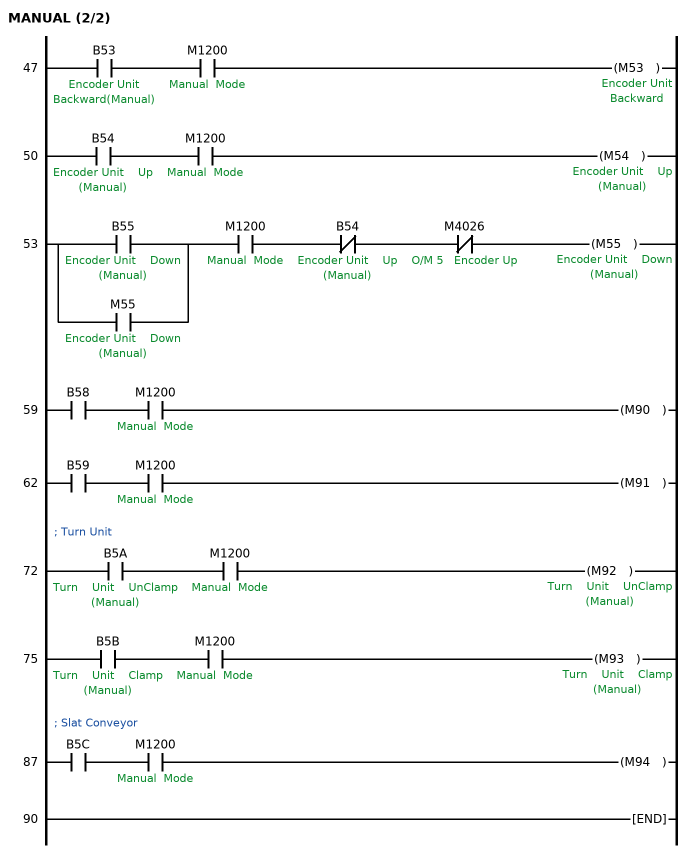
[picture p24: ladder of MANUAL, rungs at steps 47 to 90]
47    LD      B53  ; Encoder Unit    Backward(Manual)
      AND     M1200  ; Manual  Mode
      OUT     M53  ; Encoder Unit    Backward
50    LD      B54  ; Encoder Unit    Up      (Manual)
      AND     M1200  ; Manual  Mode
      OUT     M54  ; Encoder Unit    Up      (Manual)
53    LD      B55  ; Encoder Unit    Down    (Manual)
      OR      M55  ; Encoder Unit    Down    (Manual)
      AND     M1200  ; Manual  Mode
      ANI     B54  ; Encoder Unit    Up      (Manual)
      ANI     M4026  ; O/M 5   Encoder Up
      OUT     M55  ; Encoder Unit    Down    (Manual)
59    LD      B58
      AND     M1200  ; Manual  Mode
      OUT     M90
62    LD      B59
      AND     M1200  ; Manual  Mode
      OUT     M91
; Turn Unit
72    LD      B5A  ; Turn    Unit    UnClamp (Manual)
      AND     M1200  ; Manual  Mode
      OUT     M92  ; Turn    Unit    UnClamp (Manual)
75    LD      B5B  ; Turn    Unit    Clamp   (Manual)
      AND     M1200  ; Manual  Mode
      OUT     M93  ; Turn    Unit    Clamp   (Manual)
; Slat Conveyor
87    LD      B5C
      AND     M1200  ; Manual  Mode
      OUT     M94
90    END
END_PROGRAM

PROGRAM ORIGIN
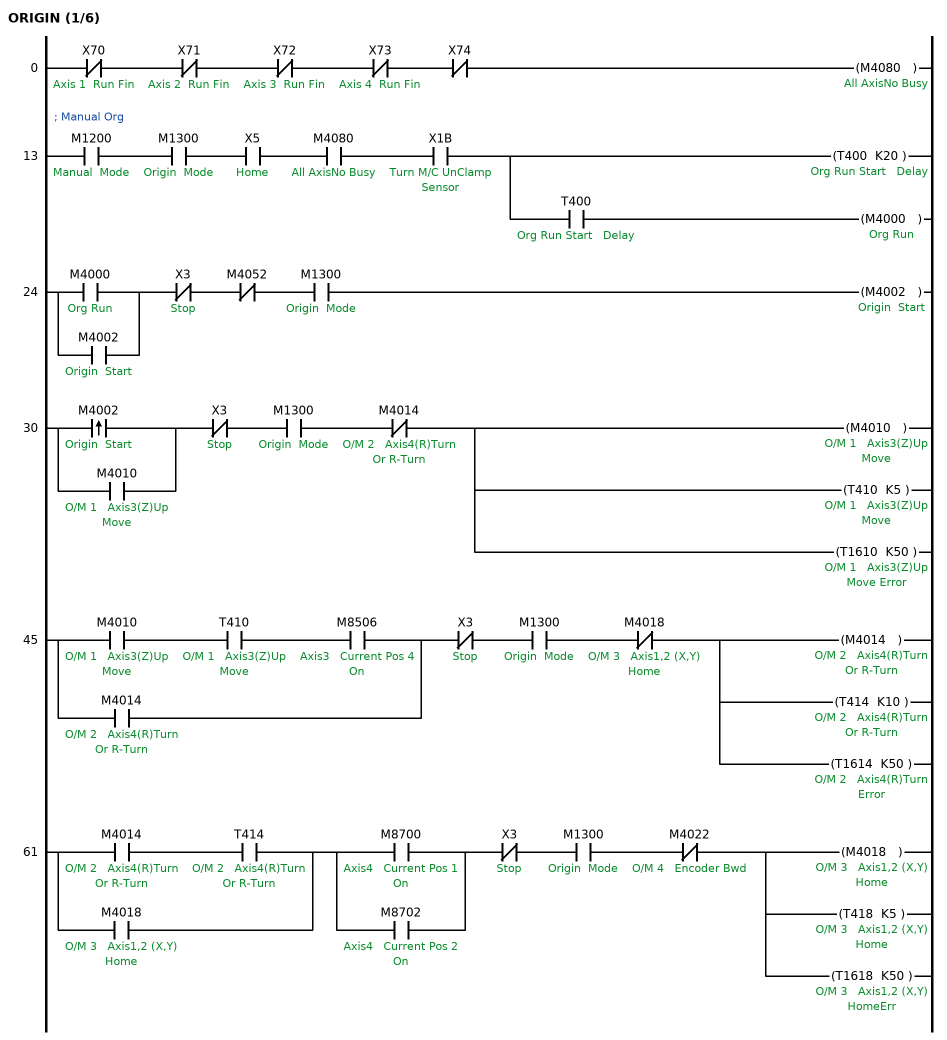
0     LDI     X70  ; Axis 1  Run Fin
      ANI     X71  ; Axis 2  Run Fin
      ANI     X72  ; Axis 3  Run Fin
      ANI     X73  ; Axis 4  Run Fin
      ANI     X74
      OUT     M4080  ; All AxisNo Busy
; Manual Org
13    LD      M1200  ; Manual  Mode
      AND     M1300  ; Origin  Mode
      AND     X5  ; Home
      AND     M4080  ; All AxisNo Busy
      AND     X1B  ; Turn M/C UnClamp Sensor
      OUT     T400 K20  ; Org Run Start   Delay
      AND     T400  ; Org Run Start   Delay
      OUT     M4000  ; Org Run
24    LD      M4000  ; Org Run
      OR      M4002  ; Origin  Start
      ANI     X3  ; Stop
      ANI     M4052
      AND     M1300  ; Origin  Mode
      OUT     M4002  ; Origin  Start
30    LDP     M4002  ; Origin  Start
      OR      M4010  ; O/M 1   Axis3(Z)Up Move
      ANI     X3  ; Stop
      AND     M1300  ; Origin  Mode
      ANI     M4014  ; O/M 2   Axis4(R)Turn Or R-Turn
      OUT     M4010  ; O/M 1   Axis3(Z)Up Move
      OUT     T410 K5  ; O/M 1   Axis3(Z)Up Move
      OUT     T1610 K50  ; O/M 1   Axis3(Z)Up Move Error
45    LD      M4010  ; O/M 1   Axis3(Z)Up Move
      AND     T410  ; O/M 1   Axis3(Z)Up Move
      AND     M8506  ; Axis3   Current Pos 4 On
      OR      M4014  ; O/M 2   Axis4(R)Turn Or R-Turn
      ANI     X3  ; Stop
      AND     M1300  ; Origin  Mode
      ANI     M4018  ; O/M 3   Axis1,2 (X,Y)   Home
      OUT     M4014  ; O/M 2   Axis4(R)Turn Or R-Turn
      OUT     T414 K10  ; O/M 2   Axis4(R)Turn Or R-Turn
      OUT     T1614 K50  ; O/M 2   Axis4(R)Turn    Error
61    LD      M4014  ; O/M 2   Axis4(R)Turn Or R-Turn
      AND     T414  ; O/M 2   Axis4(R)Turn Or R-Turn
      OR      M4018  ; O/M 3   Axis1,2 (X,Y)   Home
      LD      M8700  ; Axis4   Current Pos 1 On
      OR      M8702  ; Axis4   Current Pos 2 On
      ANB
      ANI     X3  ; Stop
      AND     M1300  ; Origin  Mode
      ANI     M4022  ; O/M 4   Encoder Bwd
      OUT     M4018  ; O/M 3   Axis1,2 (X,Y)   Home
      OUT     T418 K5  ; O/M 3   Axis1,2 (X,Y)   Home
      OUT     T1618 K50  ; O/M 3   Axis1,2 (X,Y)   HomeErr
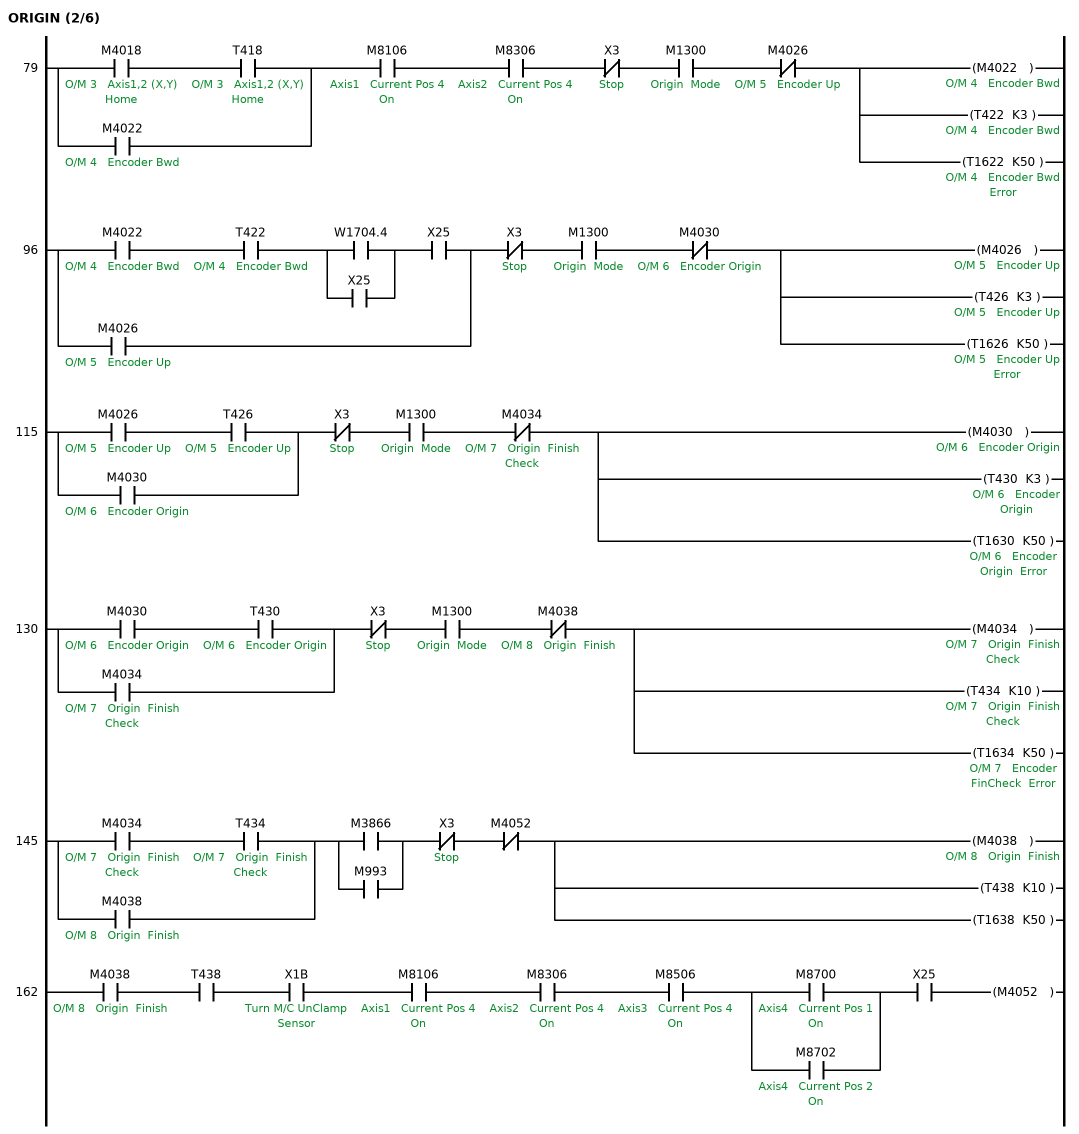
79    LD      M4018  ; O/M 3   Axis1,2 (X,Y)   Home
      AND     T418  ; O/M 3   Axis1,2 (X,Y)   Home
      OR      M4022  ; O/M 4   Encoder Bwd
      AND     M8106  ; Axis1   Current Pos 4 On
      AND     M8306  ; Axis2   Current Pos 4 On
      ANI     X3  ; Stop
      AND     M1300  ; Origin  Mode
      ANI     M4026  ; O/M 5   Encoder Up
      OUT     M4022  ; O/M 4   Encoder Bwd
      OUT     T422 K3  ; O/M 4   Encoder Bwd
      OUT     T1622 K50  ; O/M 4   Encoder Bwd     Error
96    LD      M4022  ; O/M 4   Encoder Bwd
      AND     T422  ; O/M 4   Encoder Bwd
      LD      W1704.4
      OR      X25
      ANB
      AND     X25
      OR      M4026  ; O/M 5   Encoder Up
      ANI     X3  ; Stop
      AND     M1300  ; Origin  Mode
      ANI     M4030  ; O/M 6   Encoder Origin
      OUT     M4026  ; O/M 5   Encoder Up
      OUT     T426 K3  ; O/M 5   Encoder Up
      OUT     T1626 K50  ; O/M 5   Encoder Up      Error
115   LD      M4026  ; O/M 5   Encoder Up
      AND     T426  ; O/M 5   Encoder Up
      OR      M4030  ; O/M 6   Encoder Origin
      ANI     X3  ; Stop
      AND     M1300  ; Origin  Mode
      ANI     M4034  ; O/M 7   Origin  Finish  Check
      OUT     M4030  ; O/M 6   Encoder Origin
      OUT     T430 K3  ; O/M 6   Encoder Origin
      OUT     T1630 K50  ; O/M 6   Encoder Origin  Error
130   LD      M4030  ; O/M 6   Encoder Origin
      AND     T430  ; O/M 6   Encoder Origin
      OR      M4034  ; O/M 7   Origin  Finish  Check
      ANI     X3  ; Stop
      AND     M1300  ; Origin  Mode
      ANI     M4038  ; O/M 8   Origin  Finish
      OUT     M4034  ; O/M 7   Origin  Finish  Check
      OUT     T434 K10  ; O/M 7   Origin  Finish  Check
      OUT     T1634 K50  ; O/M 7   Encoder FinCheck  Error
145   LD      M4034  ; O/M 7   Origin  Finish  Check
      AND     T434  ; O/M 7   Origin  Finish  Check
      OR      M4038  ; O/M 8   Origin  Finish
      LD      M3866
      OR      M993
      ANB
      ANI     X3  ; Stop
      ANI     M4052
      OUT     M4038  ; O/M 8   Origin  Finish
      OUT     T438 K10
      OUT     T1638 K50
162   LD      M4038  ; O/M 8   Origin  Finish
      AND     T438
      AND     X1B  ; Turn M/C UnClamp Sensor
      AND     M8106  ; Axis1   Current Pos 4 On
      AND     M8306  ; Axis2   Current Pos 4 On
      AND     M8506  ; Axis3   Current Pos 4 On
      LD      M8700  ; Axis4   Current Pos 1 On
      OR      M8702  ; Axis4   Current Pos 2 On
      ANB
      AND     X25
      OUT     M4052
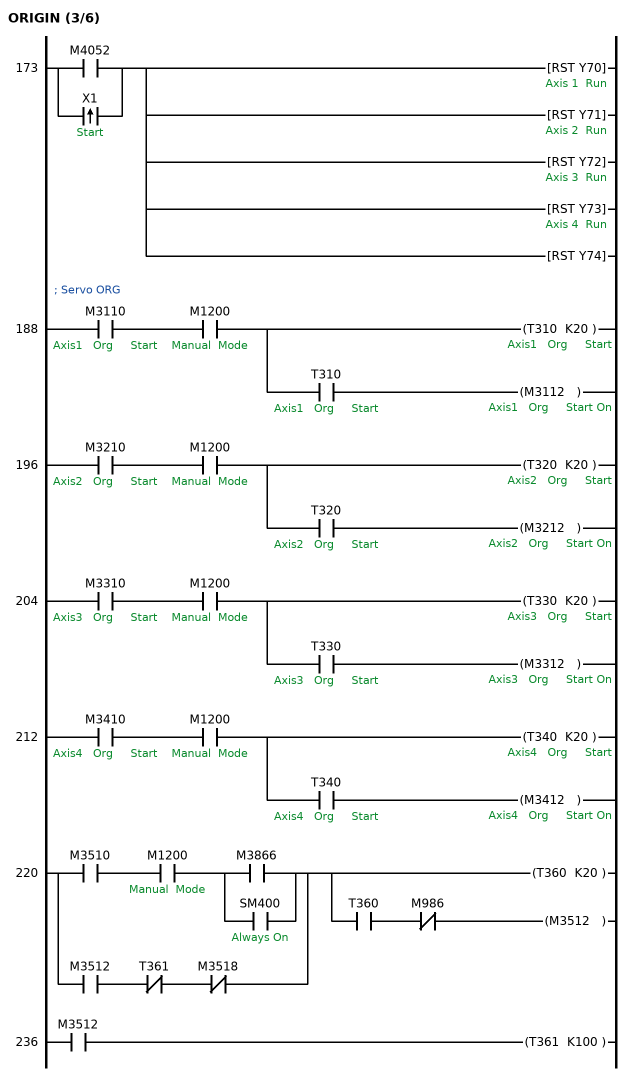
173   LD      M4052
      ORP     X1  ; Start
      RST     Y70  ; Axis 1  Run
      RST     Y71  ; Axis 2  Run
      RST     Y72  ; Axis 3  Run
      RST     Y73  ; Axis 4  Run
      RST     Y74
; Servo ORG
188   LD      M3110  ; Axis1   Org     Start
      AND     M1200  ; Manual  Mode
      OUT     T310 K20  ; Axis1   Org     Start
      AND     T310  ; Axis1   Org     Start
      OUT     M3112  ; Axis1   Org     Start On
196   LD      M3210  ; Axis2   Org     Start
      AND     M1200  ; Manual  Mode
      OUT     T320 K20  ; Axis2   Org     Start
      AND     T320  ; Axis2   Org     Start
      OUT     M3212  ; Axis2   Org     Start On
204   LD      M3310  ; Axis3   Org     Start
      AND     M1200  ; Manual  Mode
      OUT     T330 K20  ; Axis3   Org     Start
      AND     T330  ; Axis3   Org     Start
      OUT     M3312  ; Axis3   Org     Start On
212   LD      M3410  ; Axis4   Org     Start
      AND     M1200  ; Manual  Mode
      OUT     T340 K20  ; Axis4   Org     Start
      AND     T340  ; Axis4   Org     Start
      OUT     M3412  ; Axis4   Org     Start On
220   LD      M3510
      AND     M1200  ; Manual  Mode
      LD      M3866
      OR      SM400  ; Always On
      ANB
      LD      M3512
      ANI     T361
      ANI     M3518
      ORB
      OUT     T360 K20
      AND     T360
      ANI     M986
      OUT     M3512
236   LD      M3512
      OUT     T361 K100
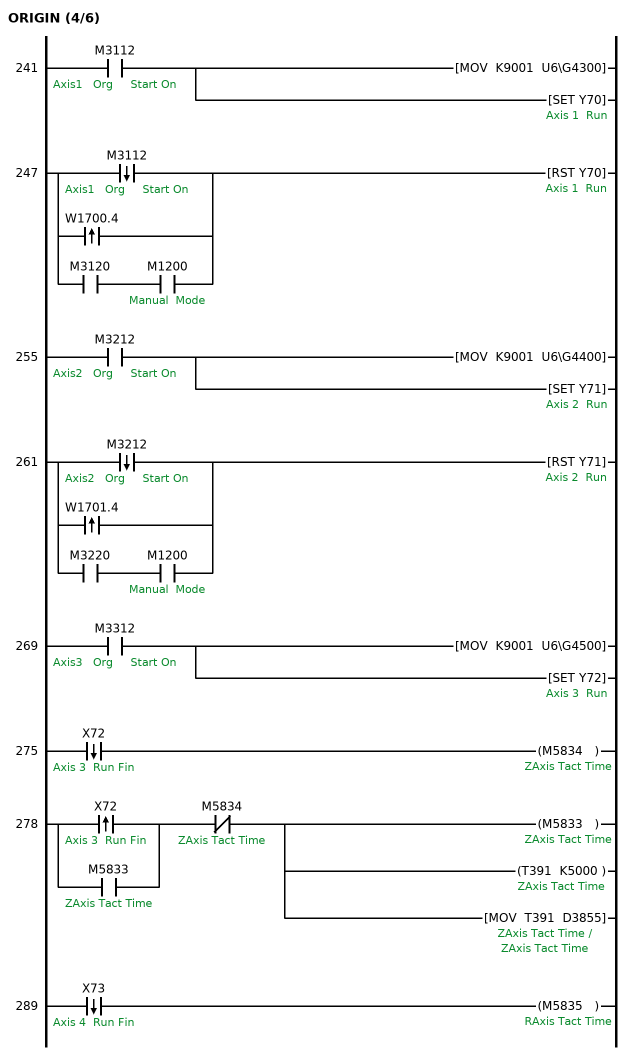
241   LD      M3112  ; Axis1   Org     Start On
      MOV     K9001 U6\G4300
      SET     Y70  ; Axis 1  Run
247   LDF     M3112  ; Axis1   Org     Start On
      ORP     W1700.4
      LD      M3120
      AND     M1200  ; Manual  Mode
      ORB
      RST     Y70  ; Axis 1  Run
255   LD      M3212  ; Axis2   Org     Start On
      MOV     K9001 U6\G4400
      SET     Y71  ; Axis 2  Run
261   LDF     M3212  ; Axis2   Org     Start On
      ORP     W1701.4
      LD      M3220
      AND     M1200  ; Manual  Mode
      ORB
      RST     Y71  ; Axis 2  Run
269   LD      M3312  ; Axis3   Org     Start On
      MOV     K9001 U6\G4500
      SET     Y72  ; Axis 3  Run
275   LDF     X72  ; Axis 3  Run Fin
      OUT     M5834  ; ZAxis Tact Time
278   LDP     X72  ; Axis 3  Run Fin
      OR      M5833  ; ZAxis Tact Time
      ANI     M5834  ; ZAxis Tact Time
      OUT     M5833  ; ZAxis Tact Time
      OUT     T391 K5000  ; ZAxis Tact Time
      MOV     T391 D3855  ; ZAxis Tact Time
289   LDF     X73  ; Axis 4  Run Fin
      OUT     M5835  ; RAxis Tact Time
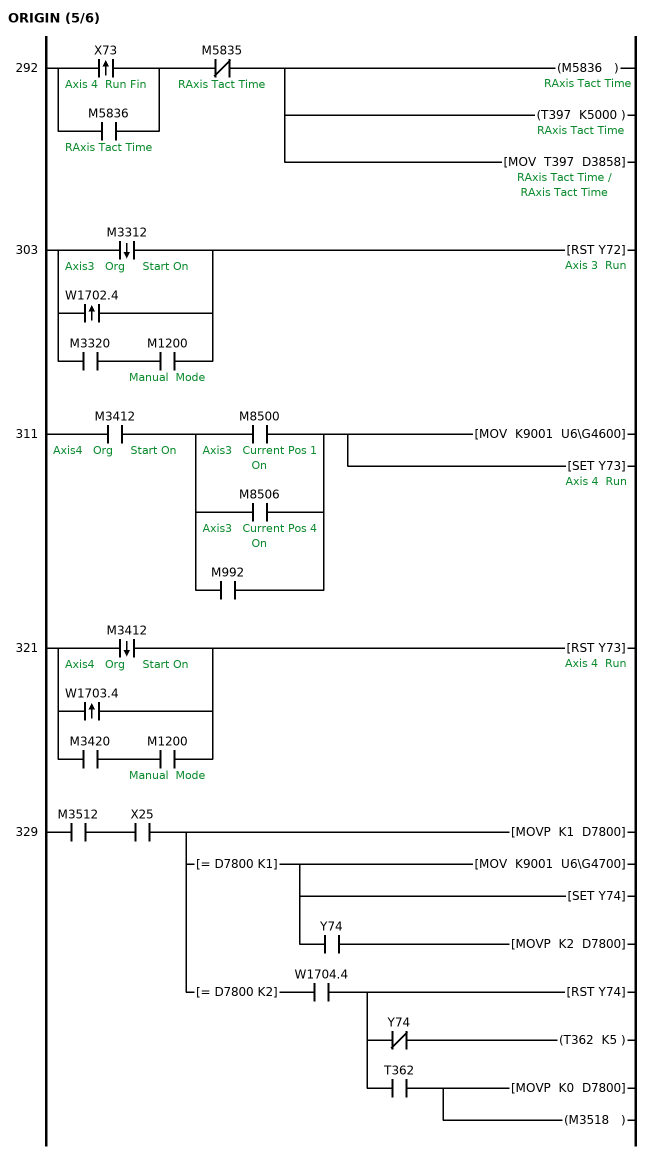
292   LDP     X73  ; Axis 4  Run Fin
      OR      M5836  ; RAxis Tact Time
      ANI     M5835  ; RAxis Tact Time
      OUT     M5836  ; RAxis Tact Time
      OUT     T397 K5000  ; RAxis Tact Time
      MOV     T397 D3858  ; RAxis Tact Time
303   LDF     M3312  ; Axis3   Org     Start On
      ORP     W1702.4
      LD      M3320
      AND     M1200  ; Manual  Mode
      ORB
      RST     Y72  ; Axis 3  Run
311   LD      M3412  ; Axis4   Org     Start On
      LD      M8500  ; Axis3   Current Pos 1 On
      OR      M8506  ; Axis3   Current Pos 4 On
      OR      M992
      ANB
      MOV     K9001 U6\G4600
      SET     Y73  ; Axis 4  Run
321   LDF     M3412  ; Axis4   Org     Start On
      ORP     W1703.4
      LD      M3420
      AND     M1200  ; Manual  Mode
      ORB
      RST     Y73  ; Axis 4  Run
329   LD      M3512
      AND     X25
      MOVP    K1 D7800
      MPS
      AND=    D7800 K1
      MOV     K9001 U6\G4700
      SET     Y74
      AND     Y74
      MOVP    K2 D7800
      MPP
      AND=    D7800 K2
      AND     W1704.4
      RST     Y74
      MPS
      ANI     Y74
      OUT     T362 K5
      MPP
      AND     T362
      MOVP    K0 D7800
      OUT     M3518
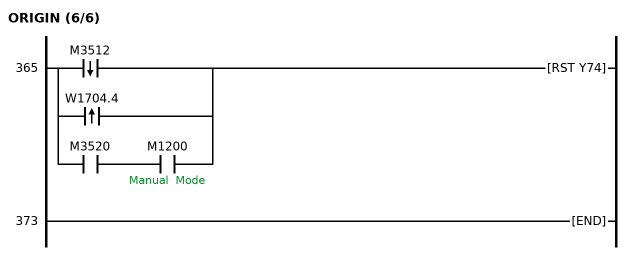
365   LDF     M3512
      ORP     W1704.4
      LD      M3520
      AND     M1200  ; Manual  Mode
      ORB
      RST     Y74
373   END
END_PROGRAM

PROGRAM POS_DATA
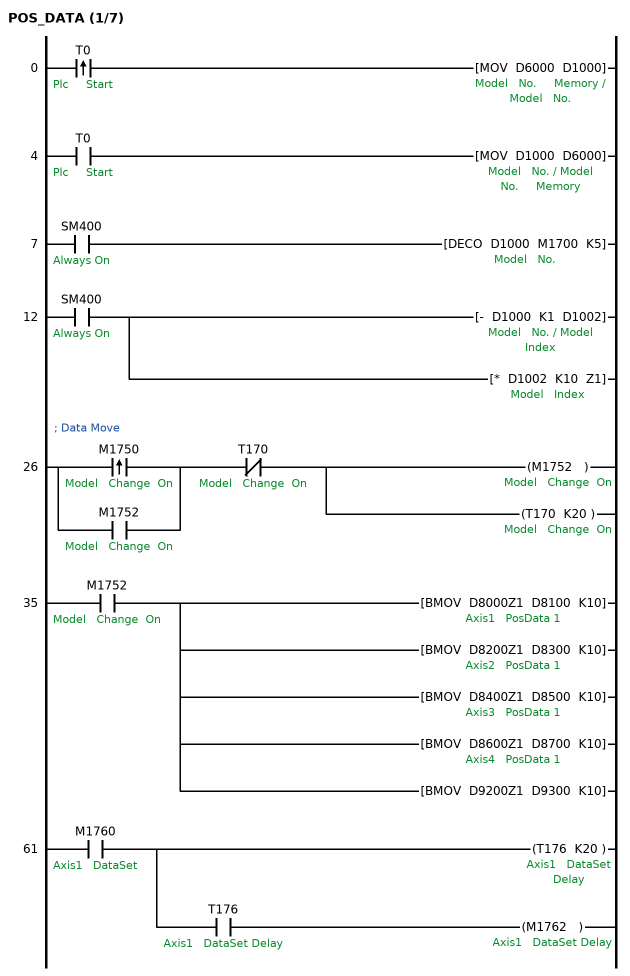
0     LDP     T0  ; Plc     Start
      MOV     D6000 D1000  ; Model   No.     Memory / Model   No.
4     LD      T0  ; Plc     Start
      MOV     D1000 D6000
7     LD      SM400  ; Always On
      DECO    D1000 M1700 K5
12    LD      SM400  ; Always On
      -       D1000 K1 D1002  ; Model   Index
      *       D1002 K10 Z1
; Data Move
26    LDP     M1750  ; Model   Change  On
      OR      M1752  ; Model   Change  On
      ANI     T170  ; Model   Change  On
      OUT     M1752  ; Model   Change  On
      OUT     T170 K20  ; Model   Change  On
35    LD      M1752  ; Model   Change  On
      BMOV    D8000Z1 D8100 K10  ; Axis1   PosData 1
      BMOV    D8200Z1 D8300 K10  ; Axis2   PosData 1
      BMOV    D8400Z1 D8500 K10  ; Axis3   PosData 1
      BMOV    D8600Z1 D8700 K10  ; Axis4   PosData 1
      BMOV    D9200Z1 D9300 K10
61    LD      M1760  ; Axis1   DataSet
      OUT     T176 K20  ; Axis1   DataSet Delay
      AND     T176  ; Axis1   DataSet Delay
      OUT     M1762  ; Axis1   DataSet Delay
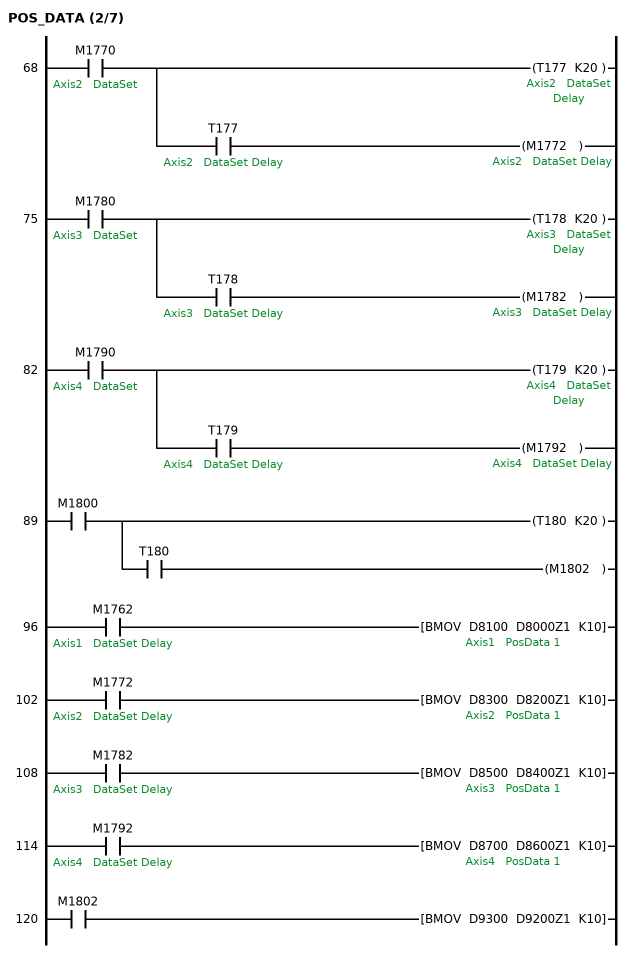
68    LD      M1770  ; Axis2   DataSet
      OUT     T177 K20  ; Axis2   DataSet Delay
      AND     T177  ; Axis2   DataSet Delay
      OUT     M1772  ; Axis2   DataSet Delay
75    LD      M1780  ; Axis3   DataSet
      OUT     T178 K20  ; Axis3   DataSet Delay
      AND     T178  ; Axis3   DataSet Delay
      OUT     M1782  ; Axis3   DataSet Delay
82    LD      M1790  ; Axis4   DataSet
      OUT     T179 K20  ; Axis4   DataSet Delay
      AND     T179  ; Axis4   DataSet Delay
      OUT     M1792  ; Axis4   DataSet Delay
89    LD      M1800
      OUT     T180 K20
      AND     T180
      OUT     M1802
96    LD      M1762  ; Axis1   DataSet Delay
      BMOV    D8100 D8000Z1 K10
102   LD      M1772  ; Axis2   DataSet Delay
      BMOV    D8300 D8200Z1 K10
108   LD      M1782  ; Axis3   DataSet Delay
      BMOV    D8500 D8400Z1 K10
114   LD      M1792  ; Axis4   DataSet Delay
      BMOV    D8700 D8600Z1 K10
120   LD      M1802
      BMOV    D9300 D9200Z1 K10
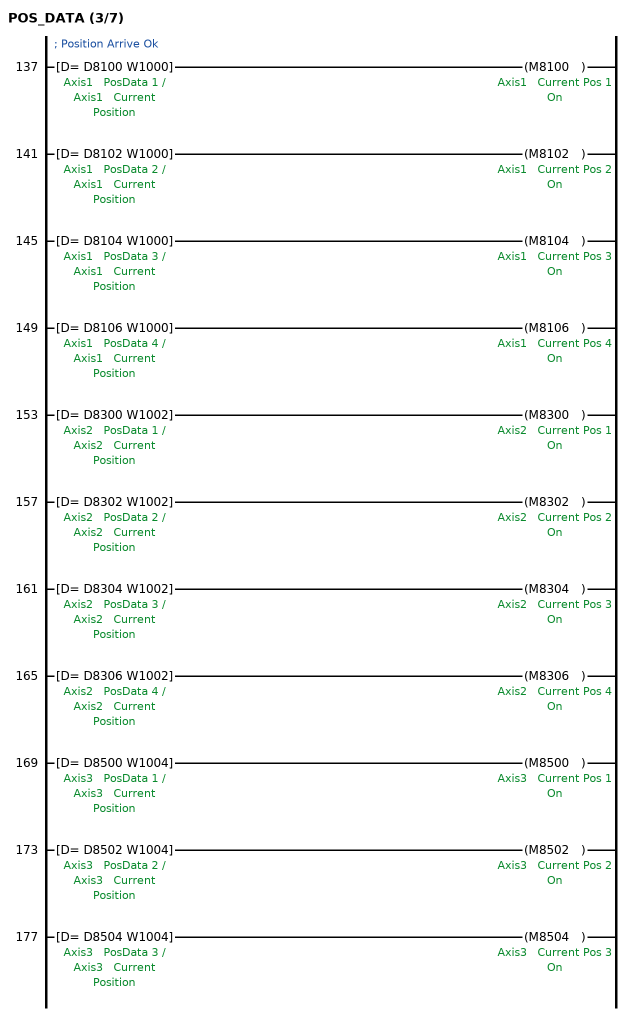
; Position Arrive Ok
137   LDD=    D8100 W1000  ; Axis1   PosData 1 / Axis1   Current Position
      OUT     M8100  ; Axis1   Current Pos 1 On
141   LDD=    D8102 W1000  ; Axis1   PosData 2 / Axis1   Current Position
      OUT     M8102  ; Axis1   Current Pos 2 On
145   LDD=    D8104 W1000  ; Axis1   PosData 3 / Axis1   Current Position
      OUT     M8104  ; Axis1   Current Pos 3 On
149   LDD=    D8106 W1000  ; Axis1   PosData 4 / Axis1   Current Position
      OUT     M8106  ; Axis1   Current Pos 4 On
153   LDD=    D8300 W1002  ; Axis2   PosData 1 / Axis2   Current Position
      OUT     M8300  ; Axis2   Current Pos 1 On
157   LDD=    D8302 W1002  ; Axis2   PosData 2 / Axis2   Current Position
      OUT     M8302  ; Axis2   Current Pos 2 On
161   LDD=    D8304 W1002  ; Axis2   PosData 3 / Axis2   Current Position
      OUT     M8304  ; Axis2   Current Pos 3 On
165   LDD=    D8306 W1002  ; Axis2   PosData 4 / Axis2   Current Position
      OUT     M8306  ; Axis2   Current Pos 4 On
169   LDD=    D8500 W1004  ; Axis3   PosData 1 / Axis3   Current Position
      OUT     M8500  ; Axis3   Current Pos 1 On
173   LDD=    D8502 W1004  ; Axis3   PosData 2 / Axis3   Current Position
      OUT     M8502  ; Axis3   Current Pos 2 On
177   LDD=    D8504 W1004  ; Axis3   PosData 3 / Axis3   Current Position
      OUT     M8504  ; Axis3   Current Pos 3 On
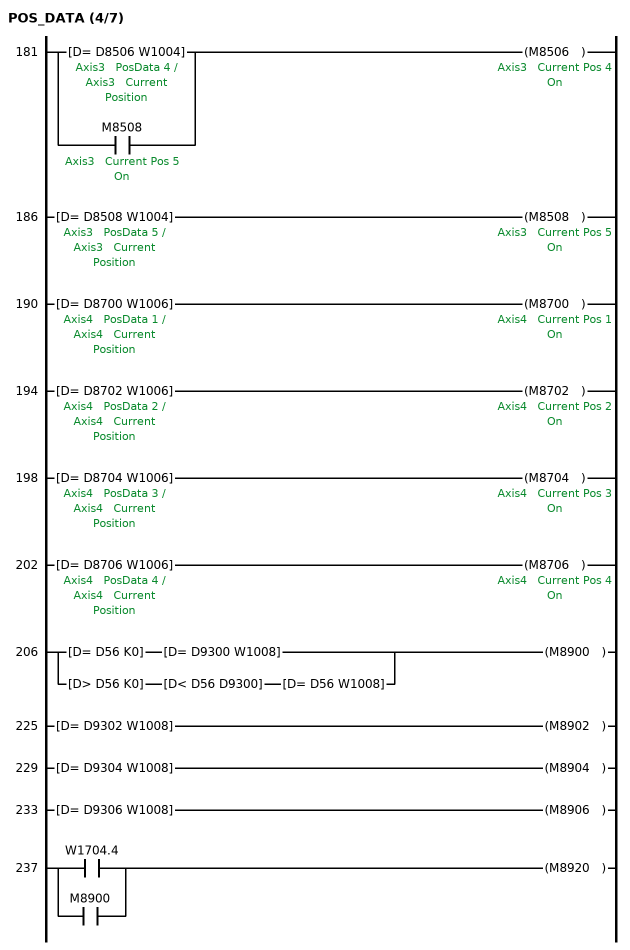
181   LDD=    D8506 W1004  ; Axis3   PosData 4 / Axis3   Current Position
      OR      M8508  ; Axis3   Current Pos 5 On
      OUT     M8506  ; Axis3   Current Pos 4 On
186   LDD=    D8508 W1004  ; Axis3   PosData 5 / Axis3   Current Position
      OUT     M8508  ; Axis3   Current Pos 5 On
190   LDD=    D8700 W1006  ; Axis4   PosData 1 / Axis4   Current Position
      OUT     M8700  ; Axis4   Current Pos 1 On
194   LDD=    D8702 W1006  ; Axis4   PosData 2 / Axis4   Current Position
      OUT     M8702  ; Axis4   Current Pos 2 On
198   LDD=    D8704 W1006  ; Axis4   PosData 3 / Axis4   Current Position
      OUT     M8704  ; Axis4   Current Pos 3 On
202   LDD=    D8706 W1006  ; Axis4   PosData 4 / Axis4   Current Position
      OUT     M8706  ; Axis4   Current Pos 4 On
206   LDD=    D56 K0
      ANDD=   D9300 W1008
      LDD>    D56 K0
      ANDD<   D56 D9300
      ANDD=   D56 W1008
      ORB
      OUT     M8900
225   LDD=    D9302 W1008
      OUT     M8902
229   LDD=    D9304 W1008
      OUT     M8904
233   LDD=    D9306 W1008
      OUT     M8906
237   LD      W1704.4
      OR      M8900
      OUT     M8920
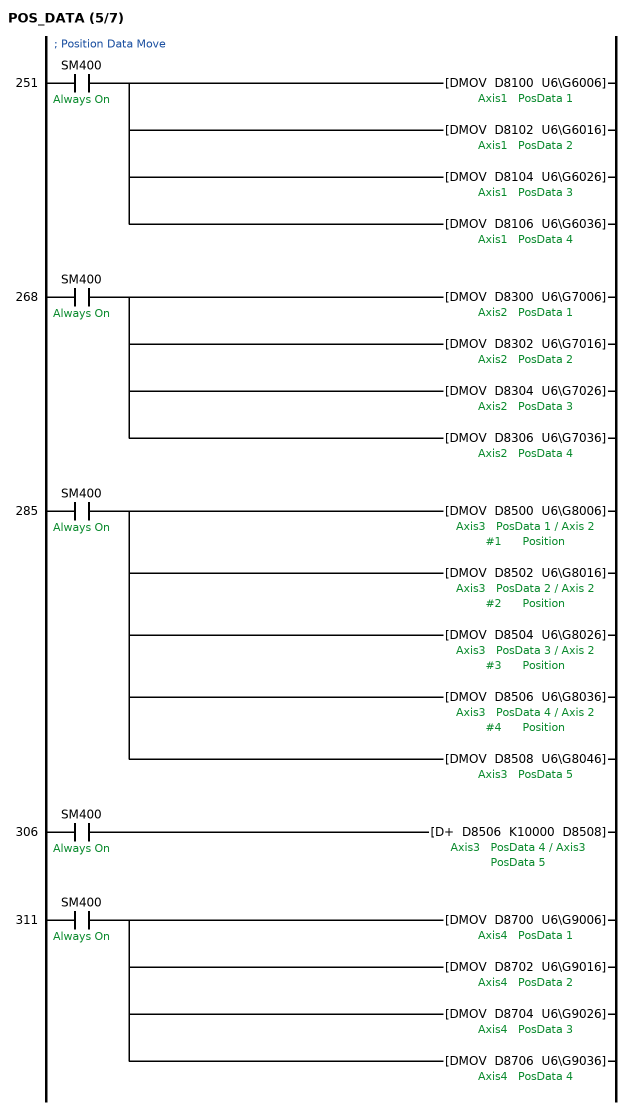
; Position Data Move
251   LD      SM400  ; Always On
      DMOV    D8100 U6\G6006
      DMOV    D8102 U6\G6016
      DMOV    D8104 U6\G6026
      DMOV    D8106 U6\G6036
268   LD      SM400  ; Always On
      DMOV    D8300 U6\G7006
      DMOV    D8302 U6\G7016
      DMOV    D8304 U6\G7026
      DMOV    D8306 U6\G7036
285   LD      SM400  ; Always On
      DMOV    D8500 U6\G8006  ; Axis 2  #1      Position
      DMOV    D8502 U6\G8016  ; Axis 2  #2      Position
      DMOV    D8504 U6\G8026  ; Axis 2  #3      Position
      DMOV    D8506 U6\G8036  ; Axis 2  #4      Position
      DMOV    D8508 U6\G8046
306   LD      SM400  ; Always On
      D+      D8506 K10000 D8508
311   LD      SM400  ; Always On
      DMOV    D8700 U6\G9006
      DMOV    D8702 U6\G9016
      DMOV    D8704 U6\G9026
      DMOV    D8706 U6\G9036
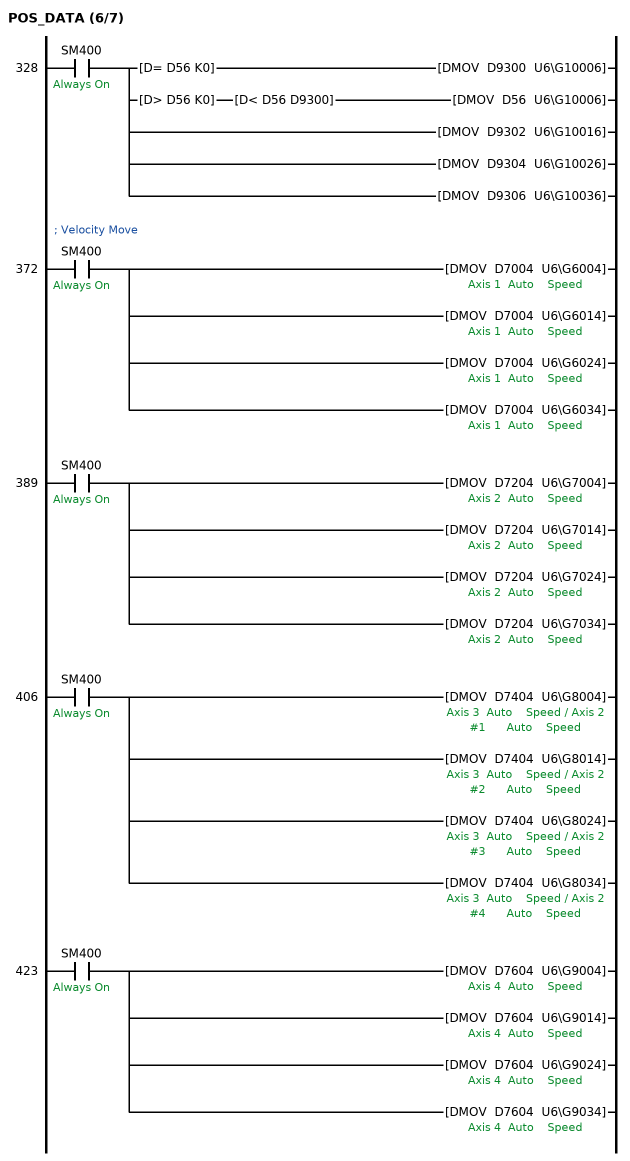
328   LD      SM400  ; Always On
      MPS
      ANDD=   D56 K0
      DMOV    D9300 U6\G10006
      MRD
      ANDD>   D56 K0
      ANDD<   D56 D9300
      DMOV    D56 U6\G10006
      MPP
      DMOV    D9302 U6\G10016
      DMOV    D9304 U6\G10026
      DMOV    D9306 U6\G10036
; Velocity Move
372   LD      SM400  ; Always On
      DMOV    D7004 U6\G6004  ; Axis 1  Auto    Speed
      DMOV    D7004 U6\G6014
      DMOV    D7004 U6\G6024
      DMOV    D7004 U6\G6034
389   LD      SM400  ; Always On
      DMOV    D7204 U6\G7004  ; Axis 2  Auto    Speed
      DMOV    D7204 U6\G7014
      DMOV    D7204 U6\G7024
      DMOV    D7204 U6\G7034
406   LD      SM400  ; Always On
      DMOV    D7404 U6\G8004  ; Axis 3  Auto    Speed / Axis 2  #1      Auto    Speed
      DMOV    D7404 U6\G8014  ; Axis 2  #2      Auto    Speed
      DMOV    D7404 U6\G8024  ; Axis 2  #3      Auto    Speed
      DMOV    D7404 U6\G8034  ; Axis 2  #4      Auto    Speed
423   LD      SM400  ; Always On
      DMOV    D7604 U6\G9004  ; Axis 4  Auto    Speed
      DMOV    D7604 U6\G9014
      DMOV    D7604 U6\G9024
      DMOV    D7604 U6\G9034
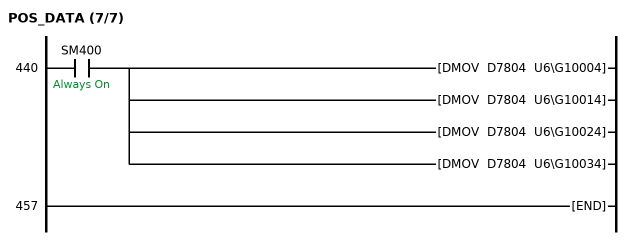
440   LD      SM400  ; Always On
      DMOV    D7804 U6\G10004
      DMOV    D7804 U6\G10014
      DMOV    D7804 U6\G10024
      DMOV    D7804 U6\G10034
457   END
END_PROGRAM

PROGRAM SERVO
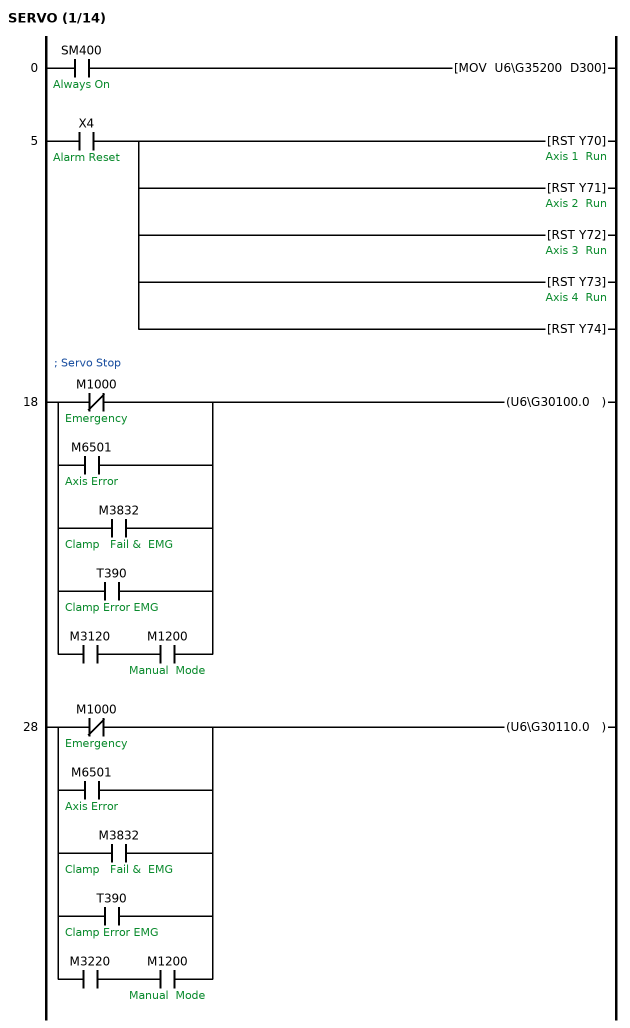
0     LD      SM400  ; Always On
      MOV     U6\G35200 D300
5     LD      X4  ; Alarm Reset
      RST     Y70  ; Axis 1  Run
      RST     Y71  ; Axis 2  Run
      RST     Y72  ; Axis 3  Run
      RST     Y73  ; Axis 4  Run
      RST     Y74
; Servo Stop
18    LDI     M1000  ; Emergency
      OR      M6501  ; Axis Error
      OR      M3832  ; Clamp   Fail &  EMG
      OR      T390  ; Clamp Error EMG
      LD      M3120
      AND     M1200  ; Manual  Mode
      ORB
      OUT     U6\G30100.0
28    LDI     M1000  ; Emergency
      OR      M6501  ; Axis Error
      OR      M3832  ; Clamp   Fail &  EMG
      OR      T390  ; Clamp Error EMG
      LD      M3220
      AND     M1200  ; Manual  Mode
      ORB
      OUT     U6\G30110.0
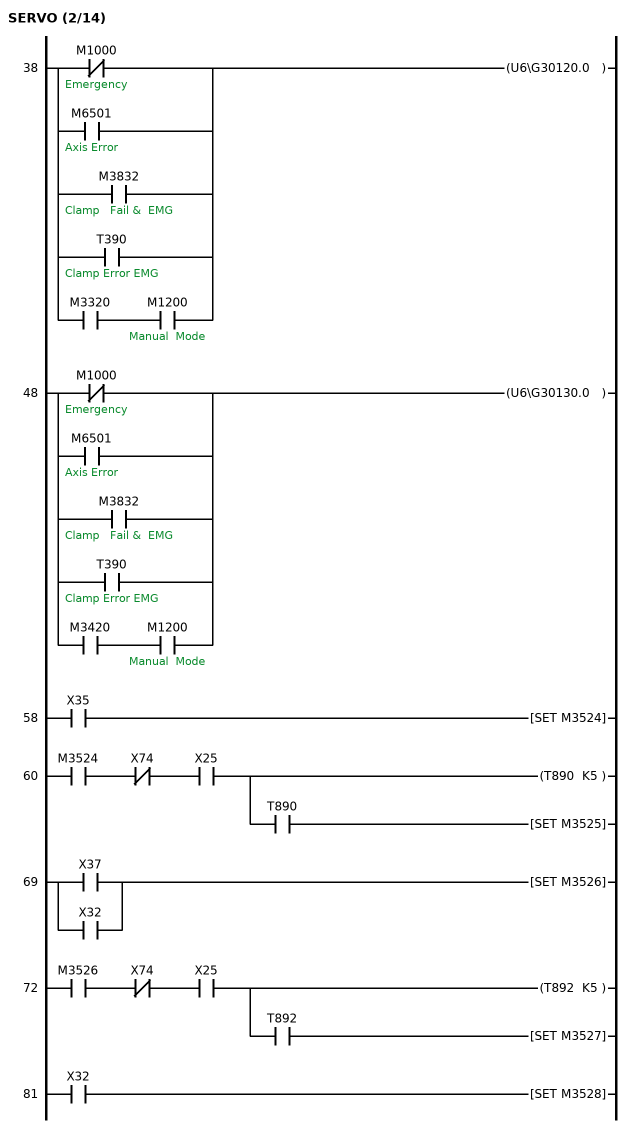
38    LDI     M1000  ; Emergency
      OR      M6501  ; Axis Error
      OR      M3832  ; Clamp   Fail &  EMG
      OR      T390  ; Clamp Error EMG
      LD      M3320
      AND     M1200  ; Manual  Mode
      ORB
      OUT     U6\G30120.0
48    LDI     M1000  ; Emergency
      OR      M6501  ; Axis Error
      OR      M3832  ; Clamp   Fail &  EMG
      OR      T390  ; Clamp Error EMG
      LD      M3420
      AND     M1200  ; Manual  Mode
      ORB
      OUT     U6\G30130.0
58    LD      X35
      SET     M3524
60    LD      M3524
      ANI     X74
      AND     X25
      OUT     T890 K5
      AND     T890
      SET     M3525
69    LD      X37
      OR      X32
      SET     M3526
72    LD      M3526
      ANI     X74
      AND     X25
      OUT     T892 K5
      AND     T892
      SET     M3527
81    LD      X32
      SET     M3528
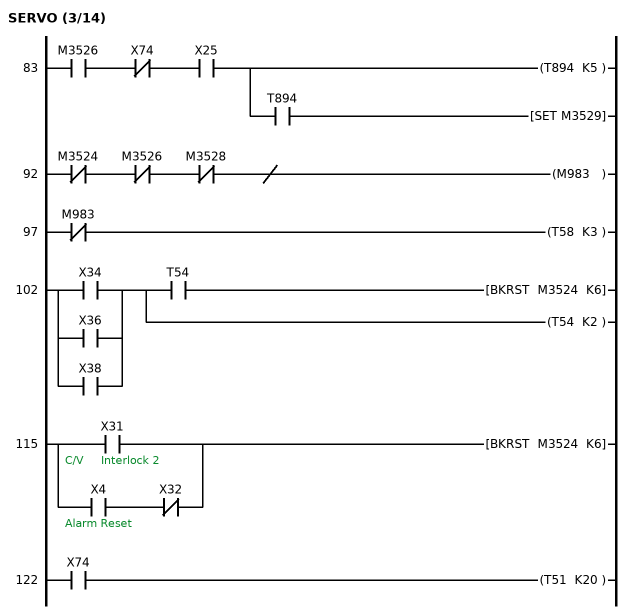
83    LD      M3526
      ANI     X74
      AND     X25
      OUT     T894 K5
      AND     T894
      SET     M3529
92    LDI     M3524
      ANI     M3526
      ANI     M3528
      INV
      OUT     M983
97    LDI     M983
      OUT     T58 K3
102   LD      X34
      OR      X36
      OR      X38
      MPS
      AND     T54
      BKRST   M3524 K6
      MPP
      OUT     T54 K2
115   LD      X31  ; C/V     Interlock 2
      LD      X4  ; Alarm Reset
      ANI     X32
      ORB
      BKRST   M3524 K6
122   LD      X74
      OUT     T51 K20
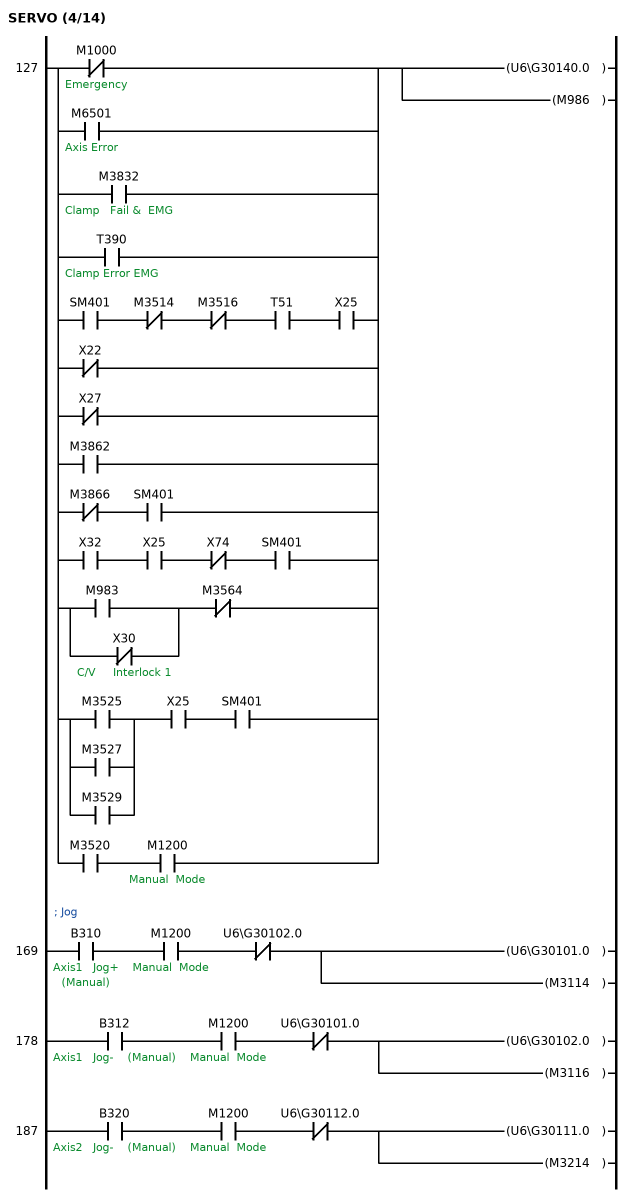
127   LDI     M1000  ; Emergency
      OR      M6501  ; Axis Error
      OR      M3832  ; Clamp   Fail &  EMG
      OR      T390  ; Clamp Error EMG
      LD      SM401
      ANI     M3514
      ANI     M3516
      AND     T51
      AND     X25
      ORB
      ORI     X22
      ORI     X27
      OR      M3862
      LDI     M3866
      AND     SM401
      ORB
      LD      X32
      AND     X25
      ANI     X74
      AND     SM401
      ORB
      LD      M983
      ORI     X30  ; C/V     Interlock 1
      ANI     M3564
      ORB
      LD      M3525
      OR      M3527
      OR      M3529
      AND     X25
      AND     SM401
      ORB
      LD      M3520
      AND     M1200  ; Manual  Mode
      ORB
      OUT     U6\G30140.0
      OUT     M986
; Jog
169   LD      B310  ; Axis1   Jog+    (Manual)
      AND     M1200  ; Manual  Mode
      ANI     U6\G30102.0
      OUT     U6\G30101.0
      OUT     M3114
178   LD      B312  ; Axis1   Jog-    (Manual)
      AND     M1200  ; Manual  Mode
      ANI     U6\G30101.0
      OUT     U6\G30102.0
      OUT     M3116
187   LD      B320  ; Axis2   Jog-    (Manual)
      AND     M1200  ; Manual  Mode
      ANI     U6\G30112.0
      OUT     U6\G30111.0
      OUT     M3214
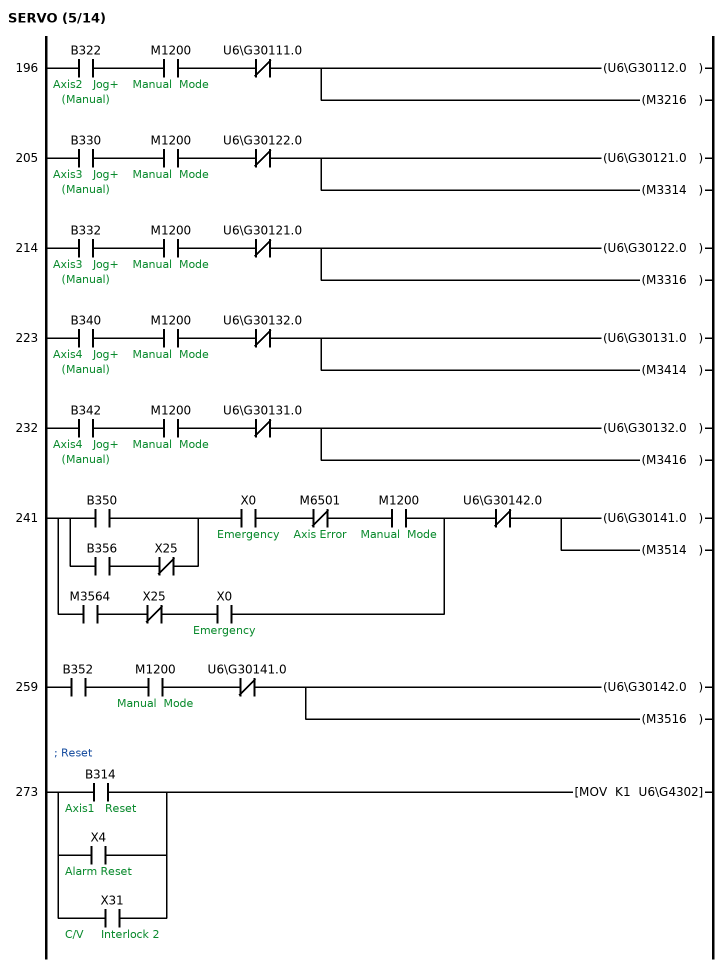
196   LD      B322  ; Axis2   Jog+    (Manual)
      AND     M1200  ; Manual  Mode
      ANI     U6\G30111.0
      OUT     U6\G30112.0
      OUT     M3216
205   LD      B330  ; Axis3   Jog+    (Manual)
      AND     M1200  ; Manual  Mode
      ANI     U6\G30122.0
      OUT     U6\G30121.0
      OUT     M3314
214   LD      B332  ; Axis3   Jog+    (Manual)
      AND     M1200  ; Manual  Mode
      ANI     U6\G30121.0
      OUT     U6\G30122.0
      OUT     M3316
223   LD      B340  ; Axis4   Jog+    (Manual)
      AND     M1200  ; Manual  Mode
      ANI     U6\G30132.0
      OUT     U6\G30131.0
      OUT     M3414
232   LD      B342  ; Axis4   Jog+    (Manual)
      AND     M1200  ; Manual  Mode
      ANI     U6\G30131.0
      OUT     U6\G30132.0
      OUT     M3416
241   LD      B350
      LD      B356
      ANI     X25
      ORB
      AND     X0  ; Emergency
      ANI     M6501  ; Axis Error
      AND     M1200  ; Manual  Mode
      LD      M3564
      ANI     X25
      AND     X0  ; Emergency
      ORB
      ANI     U6\G30142.0
      OUT     U6\G30141.0
      OUT     M3514
259   LD      B352
      AND     M1200  ; Manual  Mode
      ANI     U6\G30141.0
      OUT     U6\G30142.0
      OUT     M3516
; Reset
273   LD      B314  ; Axis1   Reset
      OR      X4  ; Alarm Reset
      OR      X31  ; C/V     Interlock 2
      MOV     K1 U6\G4302
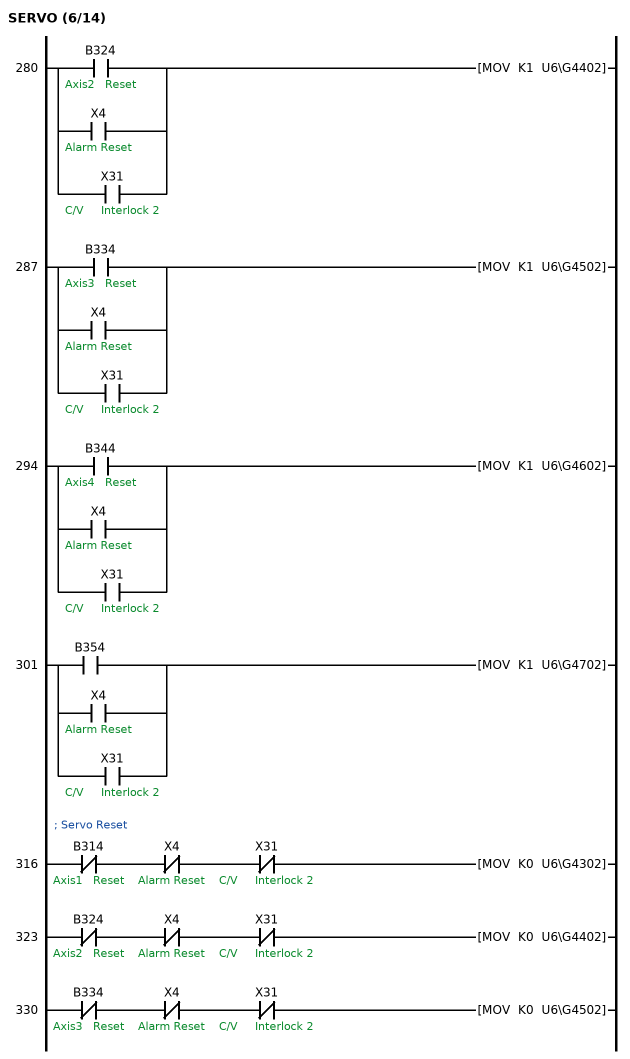
280   LD      B324  ; Axis2   Reset
      OR      X4  ; Alarm Reset
      OR      X31  ; C/V     Interlock 2
      MOV     K1 U6\G4402
287   LD      B334  ; Axis3   Reset
      OR      X4  ; Alarm Reset
      OR      X31  ; C/V     Interlock 2
      MOV     K1 U6\G4502
294   LD      B344  ; Axis4   Reset
      OR      X4  ; Alarm Reset
      OR      X31  ; C/V     Interlock 2
      MOV     K1 U6\G4602
301   LD      B354
      OR      X4  ; Alarm Reset
      OR      X31  ; C/V     Interlock 2
      MOV     K1 U6\G4702
; Servo Reset
316   LDI     B314  ; Axis1   Reset
      ANI     X4  ; Alarm Reset
      ANI     X31  ; C/V     Interlock 2
      MOV     K0 U6\G4302
323   LDI     B324  ; Axis2   Reset
      ANI     X4  ; Alarm Reset
      ANI     X31  ; C/V     Interlock 2
      MOV     K0 U6\G4402
330   LDI     B334  ; Axis3   Reset
      ANI     X4  ; Alarm Reset
      ANI     X31  ; C/V     Interlock 2
      MOV     K0 U6\G4502
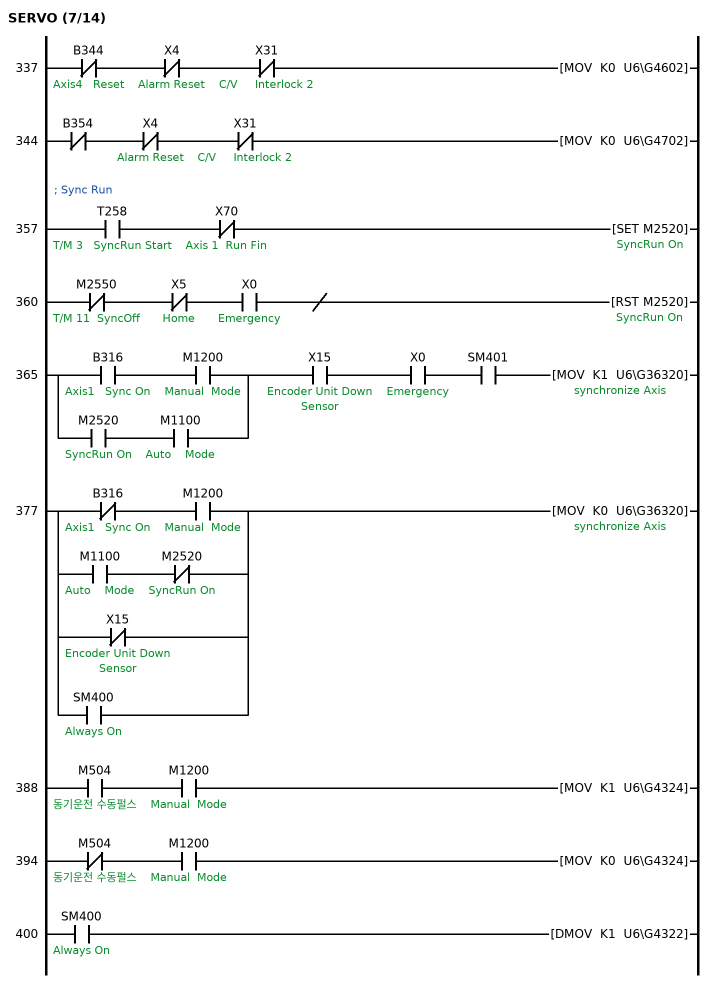
337   LDI     B344  ; Axis4   Reset
      ANI     X4  ; Alarm Reset
      ANI     X31  ; C/V     Interlock 2
      MOV     K0 U6\G4602
344   LDI     B354
      ANI     X4  ; Alarm Reset
      ANI     X31  ; C/V     Interlock 2
      MOV     K0 U6\G4702
; Sync Run
357   LD      T258  ; T/M 3   SyncRun Start
      ANI     X70  ; Axis 1  Run Fin
      SET     M2520  ; SyncRun On
360   LDI     M2550  ; T/M 11  SyncOff
      ANI     X5  ; Home
      AND     X0  ; Emergency
      INV
      RST     M2520  ; SyncRun On
365   LD      B316  ; Axis1   Sync On
      AND     M1200  ; Manual  Mode
      LD      M2520  ; SyncRun On
      AND     M1100  ; Auto    Mode
      ORB
      AND     X15  ; Encoder Unit Down Sensor
      AND     X0  ; Emergency
      AND     SM401
      MOV     K1 U6\G36320  ; synchronize Axis
377   LDI     B316  ; Axis1   Sync On
      AND     M1200  ; Manual  Mode
      LD      M1100  ; Auto    Mode
      ANI     M2520  ; SyncRun On
      ORB
      ORI     X15  ; Encoder Unit Down Sensor
      OR      SM400  ; Always On
      MOV     K0 U6\G36320
388   LD      M504  ; 동기운전 수동펄스
      AND     M1200  ; Manual  Mode
      MOV     K1 U6\G4324
394   LDI     M504  ; 동기운전 수동펄스
      AND     M1200  ; Manual  Mode
      MOV     K0 U6\G4324
400   LD      SM400  ; Always On
      DMOV    K1 U6\G4322
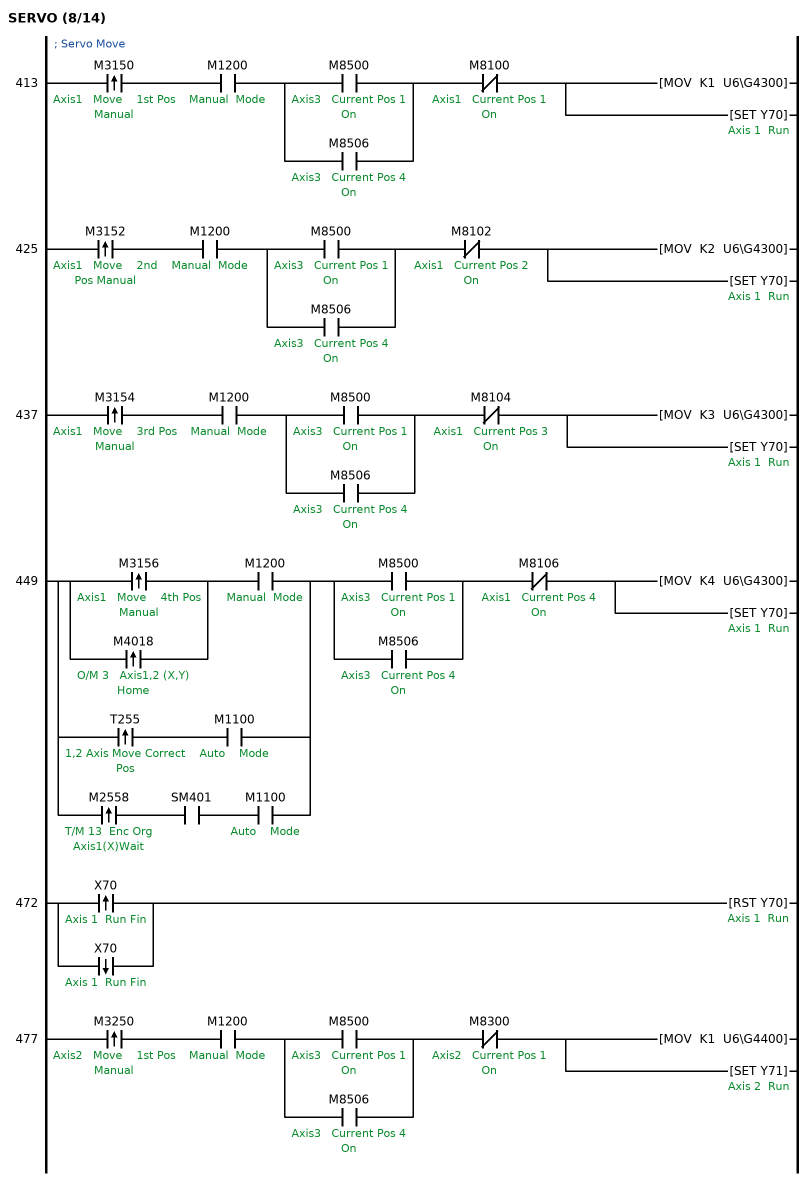
; Servo Move
413   LDP     M3150  ; Axis1   Move    1st Pos Manual
      AND     M1200  ; Manual  Mode
      LD      M8500  ; Axis3   Current Pos 1 On
      OR      M8506  ; Axis3   Current Pos 4 On
      ANB
      ANI     M8100  ; Axis1   Current Pos 1 On
      MOV     K1 U6\G4300
      SET     Y70  ; Axis 1  Run
425   LDP     M3152  ; Axis1   Move    2nd Pos Manual
      AND     M1200  ; Manual  Mode
      LD      M8500  ; Axis3   Current Pos 1 On
      OR      M8506  ; Axis3   Current Pos 4 On
      ANB
      ANI     M8102  ; Axis1   Current Pos 2 On
      MOV     K2 U6\G4300
      SET     Y70  ; Axis 1  Run
437   LDP     M3154  ; Axis1   Move    3rd Pos Manual
      AND     M1200  ; Manual  Mode
      LD      M8500  ; Axis3   Current Pos 1 On
      OR      M8506  ; Axis3   Current Pos 4 On
      ANB
      ANI     M8104  ; Axis1   Current Pos 3 On
      MOV     K3 U6\G4300
      SET     Y70  ; Axis 1  Run
449   LDP     M3156  ; Axis1   Move    4th Pos Manual
      ORP     M4018  ; O/M 3   Axis1,2 (X,Y)   Home
      AND     M1200  ; Manual  Mode
      LDP     T255  ; 1,2 Axis Move Correct Pos
      AND     M1100  ; Auto    Mode
      ORB
      LDP     M2558  ; T/M 13  Enc Org Axis1(X)Wait
      AND     SM401
      AND     M1100  ; Auto    Mode
      ORB
      LD      M8500  ; Axis3   Current Pos 1 On
      OR      M8506  ; Axis3   Current Pos 4 On
      ANB
      ANI     M8106  ; Axis1   Current Pos 4 On
      MOV     K4 U6\G4300
      SET     Y70  ; Axis 1  Run
472   LDP     X70  ; Axis 1  Run Fin
      ORF     X70  ; Axis 1  Run Fin
      RST     Y70  ; Axis 1  Run
477   LDP     M3250  ; Axis2   Move    1st Pos Manual
      AND     M1200  ; Manual  Mode
      LD      M8500  ; Axis3   Current Pos 1 On
      OR      M8506  ; Axis3   Current Pos 4 On
      ANB
      ANI     M8300  ; Axis2   Current Pos 1 On
      MOV     K1 U6\G4400
      SET     Y71  ; Axis 2  Run
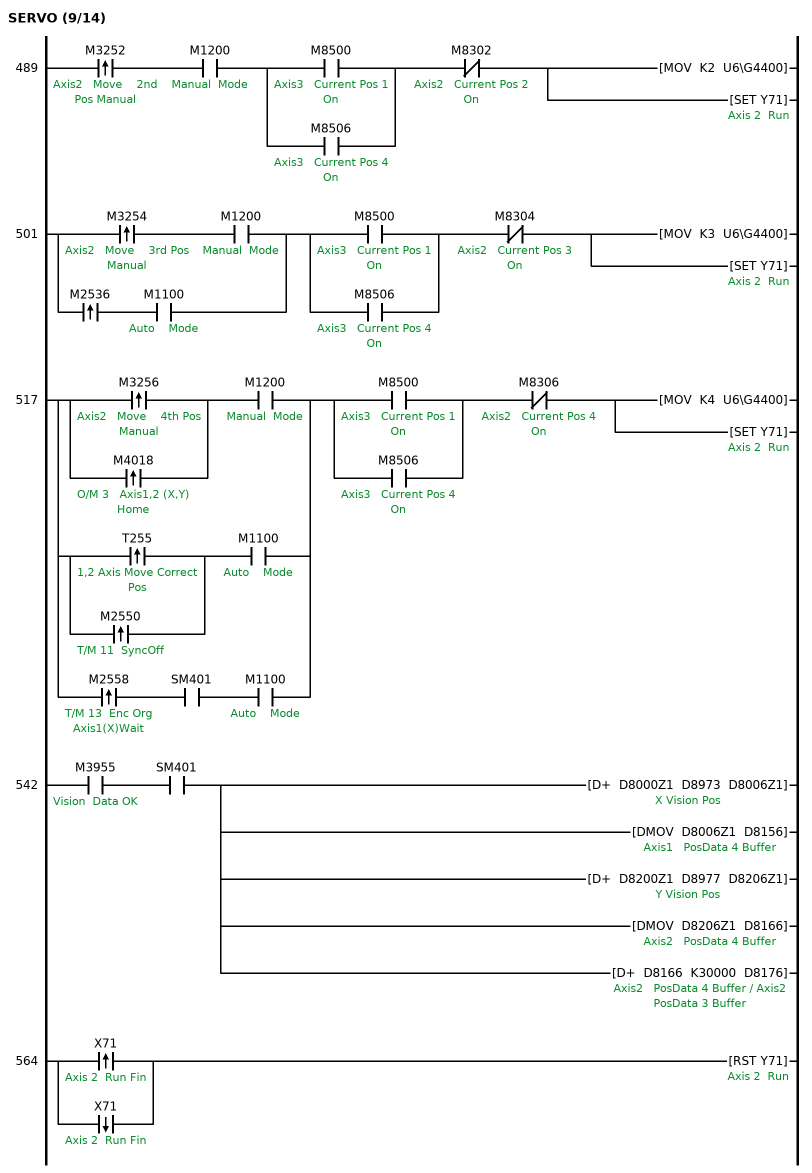
489   LDP     M3252  ; Axis2   Move    2nd Pos Manual
      AND     M1200  ; Manual  Mode
      LD      M8500  ; Axis3   Current Pos 1 On
      OR      M8506  ; Axis3   Current Pos 4 On
      ANB
      ANI     M8302  ; Axis2   Current Pos 2 On
      MOV     K2 U6\G4400
      SET     Y71  ; Axis 2  Run
501   LDP     M3254  ; Axis2   Move    3rd Pos Manual
      AND     M1200  ; Manual  Mode
      LDP     M2536
      AND     M1100  ; Auto    Mode
      ORB
      LD      M8500  ; Axis3   Current Pos 1 On
      OR      M8506  ; Axis3   Current Pos 4 On
      ANB
      ANI     M8304  ; Axis2   Current Pos 3 On
      MOV     K3 U6\G4400
      SET     Y71  ; Axis 2  Run
517   LDP     M3256  ; Axis2   Move    4th Pos Manual
      ORP     M4018  ; O/M 3   Axis1,2 (X,Y)   Home
      AND     M1200  ; Manual  Mode
      LDP     T255  ; 1,2 Axis Move Correct Pos
      ORP     M2550  ; T/M 11  SyncOff
      AND     M1100  ; Auto    Mode
      ORB
      LDP     M2558  ; T/M 13  Enc Org Axis1(X)Wait
      AND     SM401
      AND     M1100  ; Auto    Mode
      ORB
      LD      M8500  ; Axis3   Current Pos 1 On
      OR      M8506  ; Axis3   Current Pos 4 On
      ANB
      ANI     M8306  ; Axis2   Current Pos 4 On
      MOV     K4 U6\G4400
      SET     Y71  ; Axis 2  Run
542   LD      M3955  ; Vision  Data OK
      AND     SM401
      D+      D8000Z1 D8973 D8006Z1  ; X Vision Pos
      DMOV    D8006Z1 D8156  ; Axis1   PosData 4 Buffer
      D+      D8200Z1 D8977 D8206Z1  ; Y Vision Pos
      DMOV    D8206Z1 D8166  ; Axis2   PosData 4 Buffer
      D+      D8166 K30000 D8176  ; Axis2   PosData 3 Buffer
564   LDP     X71  ; Axis 2  Run Fin
      ORF     X71  ; Axis 2  Run Fin
      RST     Y71  ; Axis 2  Run
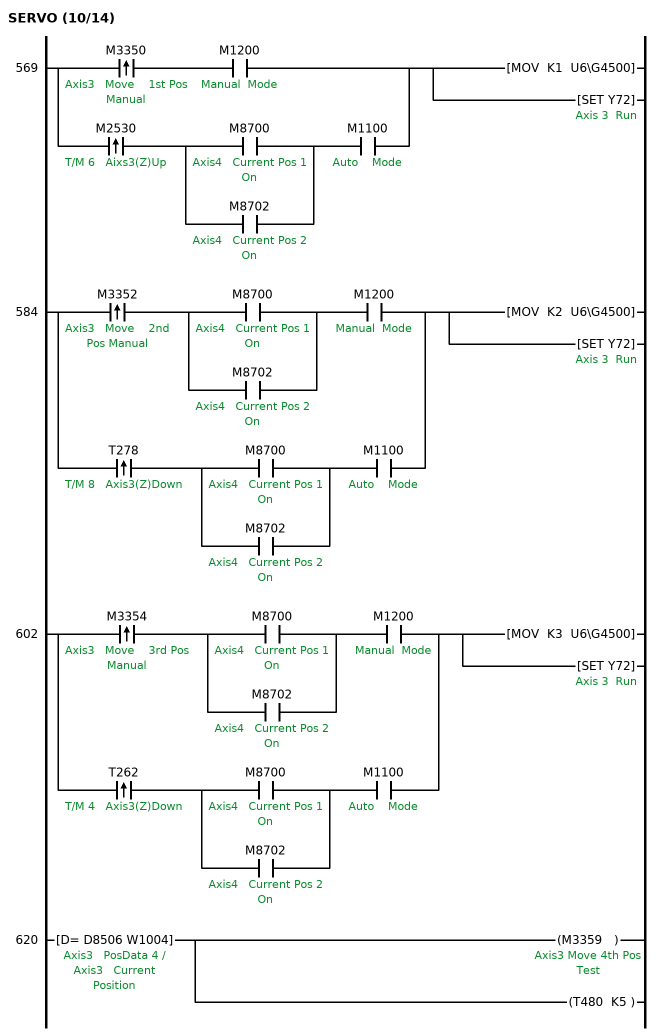
569   LDP     M3350  ; Axis3   Move    1st Pos Manual
      AND     M1200  ; Manual  Mode
      LDP     M2530  ; T/M 6   Aixs3(Z)Up
      LD      M8700  ; Axis4   Current Pos 1 On
      OR      M8702  ; Axis4   Current Pos 2 On
      ANB
      AND     M1100  ; Auto    Mode
      ORB
      MOV     K1 U6\G4500
      SET     Y72  ; Axis 3  Run
584   LDP     M3352  ; Axis3   Move    2nd Pos Manual
      LD      M8700  ; Axis4   Current Pos 1 On
      OR      M8702  ; Axis4   Current Pos 2 On
      ANB
      AND     M1200  ; Manual  Mode
      LDP     T278  ; T/M 8   Axis3(Z)Down
      LD      M8700  ; Axis4   Current Pos 1 On
      OR      M8702  ; Axis4   Current Pos 2 On
      ANB
      AND     M1100  ; Auto    Mode
      ORB
      MOV     K2 U6\G4500
      SET     Y72  ; Axis 3  Run
602   LDP     M3354  ; Axis3   Move    3rd Pos Manual
      LD      M8700  ; Axis4   Current Pos 1 On
      OR      M8702  ; Axis4   Current Pos 2 On
      ANB
      AND     M1200  ; Manual  Mode
      LDP     T262  ; T/M 4   Axis3(Z)Down
      LD      M8700  ; Axis4   Current Pos 1 On
      OR      M8702  ; Axis4   Current Pos 2 On
      ANB
      AND     M1100  ; Auto    Mode
      ORB
      MOV     K3 U6\G4500
      SET     Y72  ; Axis 3  Run
620   LDD=    D8506 W1004  ; Axis3   PosData 4 / Axis3   Current Position
      OUT     M3359  ; Axis3 Move 4th Pos Test
      OUT     T480 K5
